RESOURCE RES0 : EMB_RES_ECO
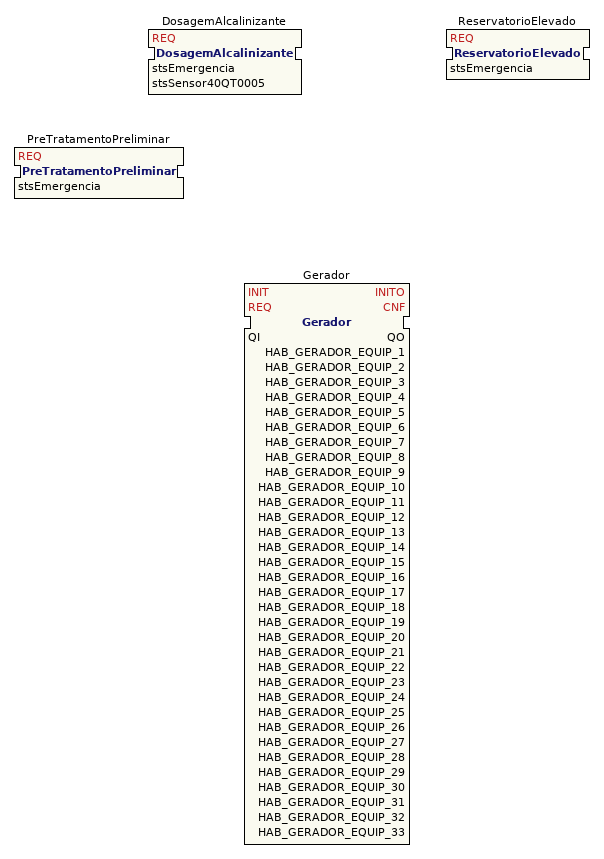
  FBS
    ReservatorioElevado : ReservatorioElevado;
    PreTratamentoPreliminar : PreTratamentoPreliminar;
    DosagemAlcalinizante : DosagemAlcalinizante;
    Gerador : Gerador;
  END_FBS
END_RESOURCE
